Xinje XCPPro project, PLC1: XC3-24 (software 3.3c)

PROGRAM Ladder

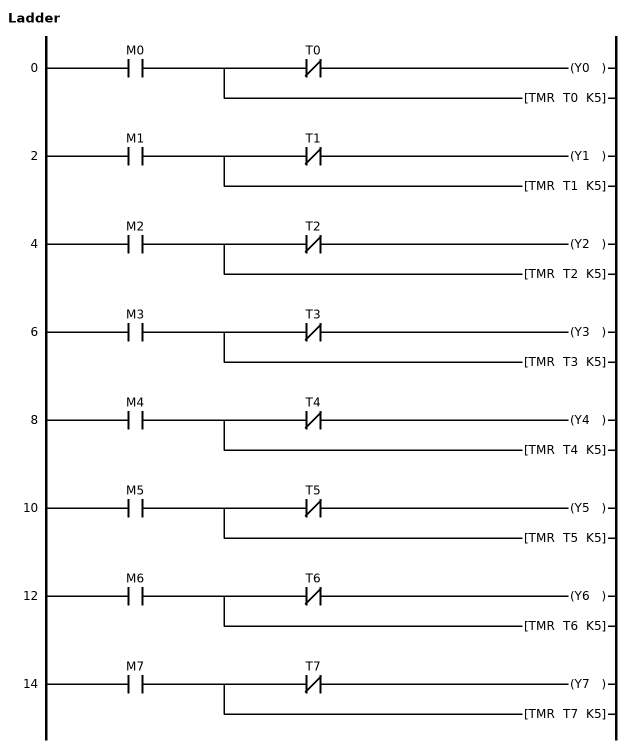
LD     M0
MPS
ANI    T0
OUT    Y0
MPP
TMR    T0 K5
LD     M1
MPS
ANI    T1
OUT    Y1
MPP
TMR    T1 K5
LD     M2
MPS
ANI    T2
OUT    Y2
MPP
TMR    T2 K5
LD     M3
MPS
ANI    T3
OUT    Y3
MPP
TMR    T3 K5
LD     M4
MPS
ANI    T4
OUT    Y4
MPP
TMR    T4 K5
LD     M5
MPS
ANI    T5
OUT    Y5
MPP
TMR    T5 K5
LD     M6
MPS
ANI    T6
OUT    Y6
MPP
TMR    T6 K5
LD     M7
MPS
ANI    T7
OUT    Y7
MPP
TMR    T7 K5